INTERFACE I_HeatingElement EXTENDS I_ComponentBase

METHOD Disable
VAR_INPUT
END_VAR
END_METHOD

METHOD Enable
VAR_INPUT
END_VAR
END_METHOD

METHOD Init
VAR_INPUT
END_VAR
END_METHOD

PROPERTY isHeating : BOOL
GET
END_GET
END_PROPERTY

METHOD PowerOff : BOOL
VAR_INPUT
END_VAR
END_METHOD

METHOD PowerOn : BOOL
VAR_INPUT
END_VAR
END_METHOD

PROPERTY State : E_State
GET
END_GET
END_PROPERTY

END_INTERFACE

(* stored: Version 1.1.0.1
   Itf I_HeatingElement: Id {38dcd78f-e4ad-41ec-b17e-8151452404c0}
   Method Disable: Id {5d720d53-a516-4a71-b3fd-ec1834526b72}
   Method Enable: Id {8d070dc6-e5b9-459f-a65f-7ad370818820}
   Method Init: Id {149fcbbe-5683-4eaa-a18f-baf6265cdab8}
   Property isHeating: Id {aa955202-bcc7-49e6-be3e-6b2adf5c56b5}
   Get Get: Id {c05e11db-a7b4-4d98-ad2a-a83f8c7d438e}
   Method PowerOff: Id {aa1b184d-5420-4f86-a1e4-c0d3db7f4e1c}
   Method PowerOn: Id {ab7f4888-a4bc-4974-9946-472316fcea99}
   Property State: Id {3e32a0d7-7de8-45d6-b51b-a5cc1b41cfc3}
   Get Get: Id {116f19d7-8cf5-4b59-962c-cda4acd476bf} *)
